KUKA KRL data list: Up14.dat

&ACCESS RVO1
&COMMENT ENTNAHME ST5085 BH1 LOW You Hua H ou
&PARAM EDITMASK = Up999[1-999]
&PARAM TEMPLATE = C:\KRC\Roboter\Template\upvorgabe
&PARAM TPVW_VERSION = 8.3.17
&PARAM DISKPATH = KRC:\R1\UPs
DEFDAT Up14
; FOLD ;%{H} %MKUKATPVW
; ENDFOLD
; interface to basic routines
EXT  BAS (BAS_COMMAND  :IN,REAL  :IN )
; interface to VW-standard routines
EXT  VW (VW_COMMAND  :IN,BOOL  :IN,REAL  :IN,REAL  :IN,REAL  :IN,REAL  :IN,BOOL  :IN,E6POS  :IN )
; interface to VW_USER - Call
EXT  VW_USER (VW_USER_CMD  :IN,INT  :IN,REAL  :IN,REAL  :IN,REAL  :IN,REAL  :IN,REAL  :IN,REAL  :IN,REAL  :IN,REAL  :IN,REAL  :IN,BOOL  :IN )
EXT  VW_USR_R (VW_USER_CMD  :IN,INT  :IN,REAL  :IN,REAL  :IN,REAL  :IN,REAL  :IN,REAL  :IN,REAL  :IN,REAL  :IN,REAL  :IN,REAL  :IN,BOOL  :IN )
EXT  IBGN (IBGN_COMMAND  :IN,BOOL  :IN,REAL  :IN,REAL  :IN,BOOL  :IN,E6POS  :OUT )
; interface select routine
EXTFCT  INT  SELECT(SUBTYPE  :IN,INT  :IN,BOOL  :IN,ARI_TYP  :IN,INT  :IN,BOOL_TYP  :IN,INT  :IN,BOOL  :IN)
INT VW_NEXT_FREE=17
INT VW_NFREE_SPS=17
INT VW_MAX_SPS=117
DECL VW_MPARA_TYP P1_D={TOOL_NO 2,BASE_NO 0,VB 100,VE 0,ACC 100,TRG_TIME 5,MOVE_TYPE #PTP_MOTION}
DECL E6POS P1={X 273.551514,Y 1212.98303,Z 954.982727,A -175.620804,B 82.2778168,C -49.8938904,S 2,T 3,E1 -518.843384,E2 0.0,E3 0.0,E4 0.0,E5 0.0,E6 0.0}
DECL VW_MPARA_TYP P2_D={TOOL_NO 2,BASE_NO 0,VB 100,VE 100,ACC 100,TRG_TIME 0,MOVE_TYPE #PTP_MOTION}
DECL E6POS P2={X 751.030212,Y 2065.62207,Z 1759.18,A 85.8736420,B 3.39197206,C -0.468862504,S 6,T 27,E1 -518.843384,E2 0.0,E3 0.0,E4 0.0,E5 0.0,E6 0.0}
DECL VW_MPARA_TYP P3_D={TOOL_NO 2,BASE_NO 0,VB 100,VE 100,ACC 100,TRG_TIME 0,MOVE_TYPE #PTP_MOTION}
DECL E6POS P3={X 793.828491,Y 1903.17297,Z 1220.16797,A 82.7425308,B 3.85024905,C -2.65520501,S 6,T 27,E1 -518.843384,E2 0.0,E3 0.0,E4 0.0,E5 0.0,E6 0.0}
DECL VW_MPARA_TYP P4_D={TOOL_NO 2,BASE_NO 0,VB 100,VE 0,ACC 100,TRG_TIME 5,MOVE_TYPE #PTP_MOTION}
DECL E6POS P4={X 756.220520,Y 2289.77808,Z 1071.79700,A 85.3607,B 3.88154602,C -0.666490376,S 6,T 27,E1 -518.843384,E2 0.0,E3 0.0,E4 0.0,E5 0.0,E6 0.0}
DECL VW_MPARA_TYP P5_D={TOOL_NO 2,BASE_NO 0,VB 400,VE 0,ACC 100,TRG_TIME 0,MOVE_TYPE #PATH_MOTION}
DECL E6POS P5={X 745.190613,Y 2600.44604,Z 1073.14099,A 85.9007187,B 3.88154411,C -0.666488588,S 6,T 27,E1 -518.843384,E2 0.0,E3 0.0,E4 0.0,E5 0.0,E6 0.0}
DECL VW_MPARA_TYP P6_D={TOOL_NO 2,BASE_NO 2,VB 400,VE 0,ACC 100,TRG_TIME 0,MOVE_TYPE #PATH_MOTION}
DECL E6POS P6={X 3330.75806,Y -754.352173,Z 1074.55396,A -4.09897,B 3.88150692,C -0.666323423,S 6,T 27,E1 -518.843384,E2 0.0,E3 0.0,E4 0.0,E5 0.0,E6 0.0}
DECL VW_MPARA_TYP P7_D={TOOL_NO 2,BASE_NO 31,VB 400,VE 100,ACC 100,TRG_TIME 0,MOVE_TYPE #PATH_MOTION}
DECL E6POS P7={X -51.4995804,Y -3.80312204,Z -1.04921496,A -1.46000E-07,B 4.20000E-08,C -2.10000E-08,S 6,T 27,E1 -518.843384,E2 0.0,E3 0.0,E4 0.0,E5 0.0,E6 0.0}
DECL VW_MPARA_TYP P8_D={TOOL_NO 2,BASE_NO 31,VB 400,VE 0,ACC 100,TRG_TIME 5,MOVE_TYPE #PATH_MOTION}
DECL E6POS P8={X -63.0451088,Y -9.65869236,Z 22.3897,A -2.35096877E-07,B -3.21929470E-08,C -4.08605167E-08,S 6,T 27,E1 -518.843384,E2 0.0,E3 0.0,E4 0.0,E5 0.0,E6 0.0}
DECL VW_MPARA_TYP P9_D={TOOL_NO 2,BASE_NO 0,VB 400,VE 0,ACC 100,TRG_TIME 0,MOVE_TYPE #PATH_MOTION}
DECL E6POS P9={X 755.152405,Y 2407.66577,Z 1104.56042,A 85.4656525,B 3.88155890,C -0.666428626,S 6,T 27,E1 -518.843384,E2 0.0,E3 0.0,E4 0.0,E5 0.0,E6 0.0}
DECL VW_MPARA_TYP P10_D={TOOL_NO 2,BASE_NO 0,VB 400,VE 0,ACC 100,TRG_TIME 0,MOVE_TYPE #PATH_MOTION}
DECL E6POS P10={X 758.783203,Y 2320.12598,Z 1120.06799,A 85.3607,B 3.88154602,C -0.666490316,S 6,T 27,E1 -518.843384,E2 0.0,E3 0.0,E4 0.0,E5 0.0,E6 0.0}
DECL VW_MPARA_TYP P11_D={TOOL_NO 2,BASE_NO 0,VB 400,VE 0,ACC 100,TRG_TIME 0,MOVE_TYPE #PATH_MOTION}
DECL E6POS P11={X 758.780,Y 2320.11401,Z 1225.52405,A 85.3609772,B 3.88154411,C -0.666295111,S 6,T 27,E1 -518.843384,E2 0.0,E3 0.0,E4 0.0,E5 0.0,E6 0.0}
DECL VW_MPARA_TYP P12_D={TOOL_NO 2,BASE_NO 0,VB 400,VE 0,ACC 100,TRG_TIME 0,MOVE_TYPE #PATH_MOTION}
DECL E6POS P12={X 758.780212,Y 2017.35,Z 1225.52405,A 85.3609772,B 3.88154292,C -0.666295528,S 6,T 27,E1 -518.843384,E2 0.0,E3 0.0,E4 0.0,E5 0.0,E6 0.0}
DECL VW_MPARA_TYP P13_D={TOOL_NO 2,BASE_NO 0,VB 400,VE 0,ACC 100,TRG_TIME 5,MOVE_TYPE #PATH_MOTION}
DECL E6POS P13={X 758.780212,Y 2017.35,Z 1225.52405,A 85.3609772,B 3.88154292,C -0.666295528,S 6,T 27,E1 -518.843384,E2 0.0,E3 0.0,E4 0.0,E5 0.0,E6 0.0}
DECL VW_MPARA_TYP P14_D={TOOL_NO 2,BASE_NO 0,VB 100,VE 100,ACC 100,TRG_TIME 0,MOVE_TYPE #PTP_MOTION}
DECL E6POS P14={X 793.828613,Y 1903.17297,Z 1220.16797,A 82.7425308,B 3.85025191,C -2.65520597,S 6,T 27,E1 -518.843384,E2 0.0,E3 0.0,E4 0.0,E5 0.0,E6 0.0}
DECL VW_MPARA_TYP P15_D={TOOL_NO 2,BASE_NO 0,VB 100,VE 100,ACC 100,TRG_TIME 0,MOVE_TYPE #PTP_MOTION}
DECL E6POS P15={X 762.078674,Y 1923.95203,Z 1713.44897,A 85.0349274,B 3.62453604,C -0.816440880,S 6,T 27,E1 -518.843384,E2 0.0,E3 0.0,E4 0.0,E5 0.0,E6 0.0}
DECL VW_MPARA_TYP P16_D={TOOL_NO 2,BASE_NO 0,VB 100,VE 0,ACC 100,TRG_TIME 5,MOVE_TYPE #PTP_MOTION}
DECL E6POS P16={X 273.551514,Y 1212.98303,Z 954.982727,A -175.620804,B 82.2778168,C -49.8938904,S 2,T 3,E1 -518.843384,E2 0.0,E3 0.0,E4 0.0,E5 0.0,E6 0.0}
ENDDAT
